// Mitsubishi GX Works2 project: Ex2   PLC: Q03UDV

PROGRAM MAIN
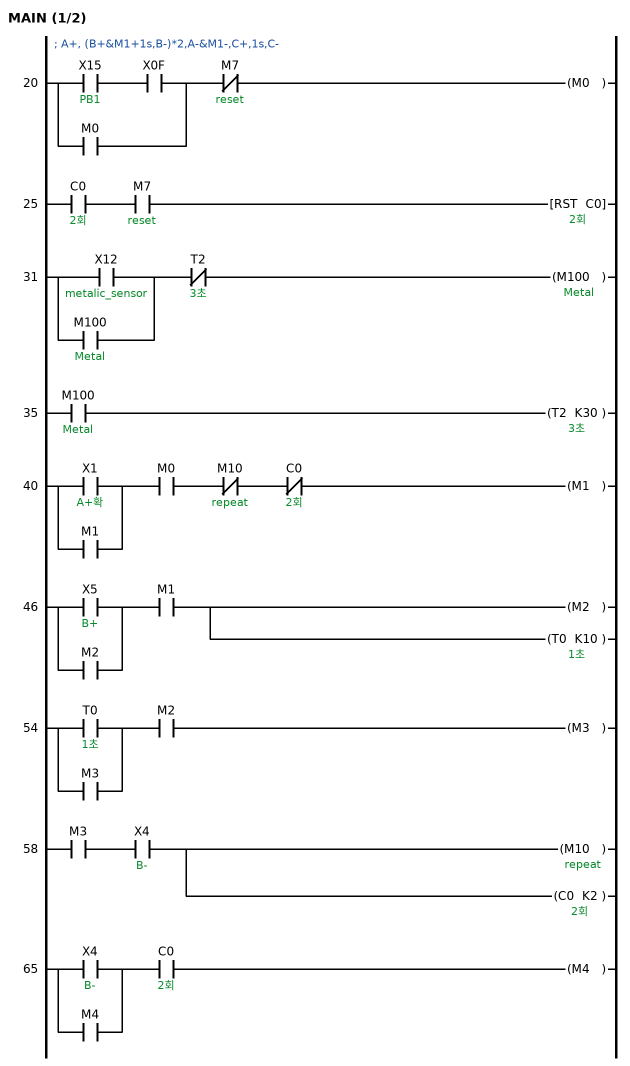
; A+, (B+&M1+1s,B-)*2,A-&M1-,C+,1s,C-
20    LD      X15  ; PB1
      AND     X0F
      OR      M0
      ANI     M7  ; reset
      OUT     M0
25    LD      C0  ; 2회
      AND     M7  ; reset
      RST     C0  ; 2회
31    LD      X12  ; metalic_sensor
      OR      M100  ; Metal
      ANI     T2  ; 3초
      OUT     M100  ; Metal
35    LD      M100  ; Metal
      OUT     T2 K30  ; 3초
40    LD      X1  ; A+확
      OR      M1
      AND     M0
      ANI     M10  ; repeat
      ANI     C0  ; 2회
      OUT     M1
46    LD      X5  ; B+
      OR      M2
      AND     M1
      OUT     M2
      OUT     T0 K10  ; 1초
54    LD      T0  ; 1초
      OR      M3
      AND     M2
      OUT     M3
58    LD      M3
      AND     X4  ; B-
      OUT     M10  ; repeat
      OUT     C0 K2  ; 2회
65    LD      X4  ; B-
      OR      M4
      AND     C0  ; 2회
      OUT     M4
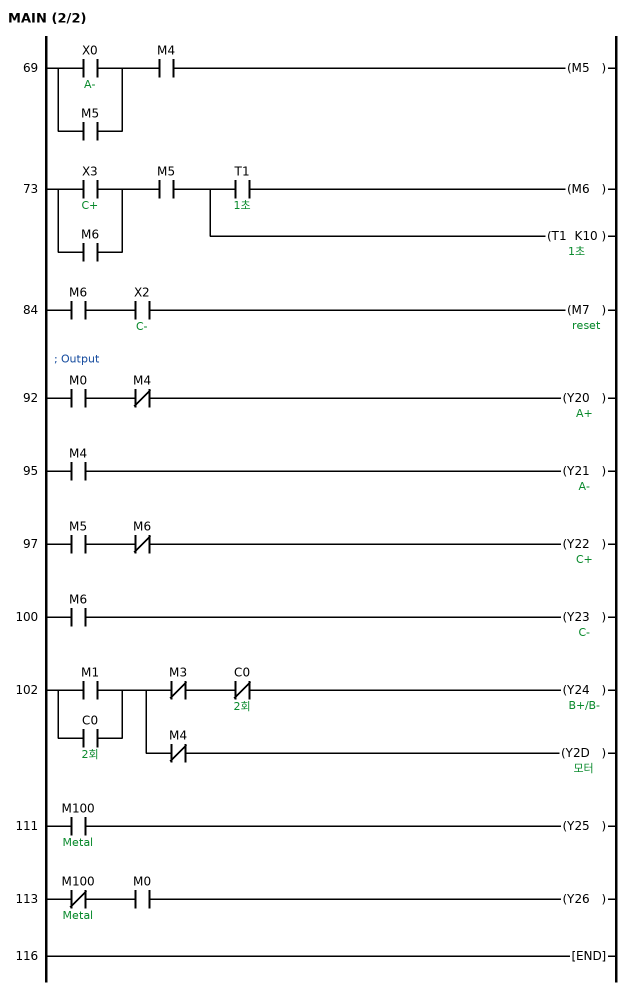
69    LD      X0  ; A-
      OR      M5
      AND     M4
      OUT     M5
73    LD      X3  ; C+
      OR      M6
      AND     M5
      MPS
      AND     T1  ; 1초
      OUT     M6
      MPP
      OUT     T1 K10  ; 1초
84    LD      M6
      AND     X2  ; C-
      OUT     M7  ; reset
; Output
92    LD      M0
      ANI     M4
      OUT     Y20  ; A+
95    LD      M4
      OUT     Y21  ; A-
97    LD      M5
      ANI     M6
      OUT     Y22  ; C+
100   LD      M6
      OUT     Y23  ; C-
102   LD      M1
      OR      C0  ; 2회
      MPS
      ANI     M3
      ANI     C0  ; 2회
      OUT     Y24  ; B+/B-
      MPP
      ANI     M4
      OUT     Y2D  ; 모터
111   LD      M100  ; Metal
      OUT     Y25
113   LDI     M100  ; Metal
      AND     M0
      OUT     Y26
116   END
END_PROGRAM

// device comments not shown above
X16  ; PB2
